TEXTLIST tlActuatorNames
  1 = 'Weighing Actuator Work' | PL: 'Weighing Actuator Work' | EN: 'Chamber Close'
  0 = 'Weighing Actuator Home' | PL: 'Weighing Actuator Home' | EN: 'Chamber Open'
  3 = 'Pusher Work' | PL: 'Pusher Work' | EN: 'Puncture Cylinder Work'
  2 = 'Pusher Home' | PL: 'Pusher Home' | EN: 'Puncture Cylinder Home'
  4 = 'Unloading Actuator Home' | PL: 'Unloading Actuator Home' | EN: 'Inlet Valve Open'
  5 = 'Unloading Actuator Work' | PL: 'Unloading Actuator Work' | EN: 'Inlet Valve Close'
   = ''
END_TEXTLIST

(* stored: Version 1.1.0.1, ProductVersion 3.1.4024.15
   TextList tlActuatorNames: Id {8c0220d9-926a-446a-9eb6-7e919a3a120d} *)
